PROGRAM PRG_TESTS

(* Instantiate test suites here. Naming convention for tests should be a suffix with _Tests.
Good practice for creating test methods is to end them with _test as well. *)
VAR
	fbSUT_Tests	: FB_SUT_Tests;
END_VAR

// Run tests in paralel
TcUnit.RUN();

// Run tests in sequence, one after the other. Uncomment if required.
// TcUnit.RUN_IN_SEQUENCE();

END_PROGRAM

(* stored: Version 1.1.0.1, ProductVersion 3.1.4024.13
   POU PRG_TESTS: Id {6e34c45a-3ca6-4d60-98ec-a84888e107c1}, SpecialFunc None *)
